# EPICS autosave request: iocBoot/generic_motors_ioc/dbSave/CCD_St_.req
%
% BURT Request File
%
% $(P)CCD:St:  CCD support
%

file assy.req ASSY=$(P)CCD:St
%%% $(P)CCD:St:H
$(P)CCD:St:dH
$(P)CCD:St:L
$(P)CCD:St:Lh
$(P)CCD:St:Lv
$(P)CCD:St:Dms
$(P)CCD:St:aV
$(P)CCD:St:mLink
file mtr1.req MTR1=$(P)CCD:mx
file mtr1.req MTR1=$(P)CCD:mus
file mtr1.req MTR1=$(P)CCD:mds
file drv1.req DRV1=$(P)CCD:X
file drv1.req DRV1=$(P)CCD:VUS
file drv1.req DRV1=$(P)CCD:VDS
file axs1.req AXS1=$(P)CCD:D
file axs1.req AXS1=$(P)CCD:2Q
